{attribute 'qualified_only'}
{attribute 'strict'}
TYPE Brewing :	// enumaration of all states for 'BrewCoffee'.
(
	OFF,
	Idle,
	HeatingWater,
	BrewCoffee
):= OFF;
END_TYPE

(* stored: Version 1.1.0.1, ProductVersion 3.1.4024.12
   DUT Brewing: Id {b25391a5-7890-4228-a169-ad2244204845} *)
